FUNCTION ASSERT : BOOL
VAR_INPUT
	passed: BOOL;
	text: STRING;
END_VAR
VAR
END_VAR

IF NOT passed THEN
	ADSLOGSTR(msgCtrlMask := ADSLOG_MSGTYPE_ERROR, msgFmtStr := 'FAILED: %s', text);
END_IF

ASSERT := passed;

END_FUNCTION

(* stored: Version 1.1.0.1, ProductVersion 3.1.4024.10
   POU ASSERT: Id {be57aea1-06b2-4728-8914-c9a75b85e098}, SpecialFunc None *)
